// TIA Portal V17 export
// export: Created 2021-12-03T08:12:56.503226Z, ExportSetting WithDefaults, DisplayName Totally Integrated Automation Portal, DisplayVersion V17, DisplayName TIA Portal Openness, DisplayVersion V17, DisplayName TIA Portal Version Control Interface, DisplayVersion V17, DisplayName STEP 7 Professional, DisplayVersion V17, DisplayName STEP 7 Safety, DisplayVersion V17, DisplayName WinCC Advanced, DisplayVersion V17
DATA_BLOCK "GDB_Gen_Ctrl"   // DB30
VERSION : 0.1
// stored: AutoNumber false, IsOnlyStoredInLoadMemory false, IsWriteProtectedInAS false
   VAR
      ServiceMode : Bool;   // Сервисный режим
      FaultReset : Bool;   // Сброс ошибок
      PeriClsAck : Bool;   // Подтверждение периметра безопасности
      Restart : Bool;
   END_VAR
BEGIN
END_DATA_BLOCK
